// Mitsubishi GX Works2 project: Final Project   PLC: Q00U

PROGRAM CLDa
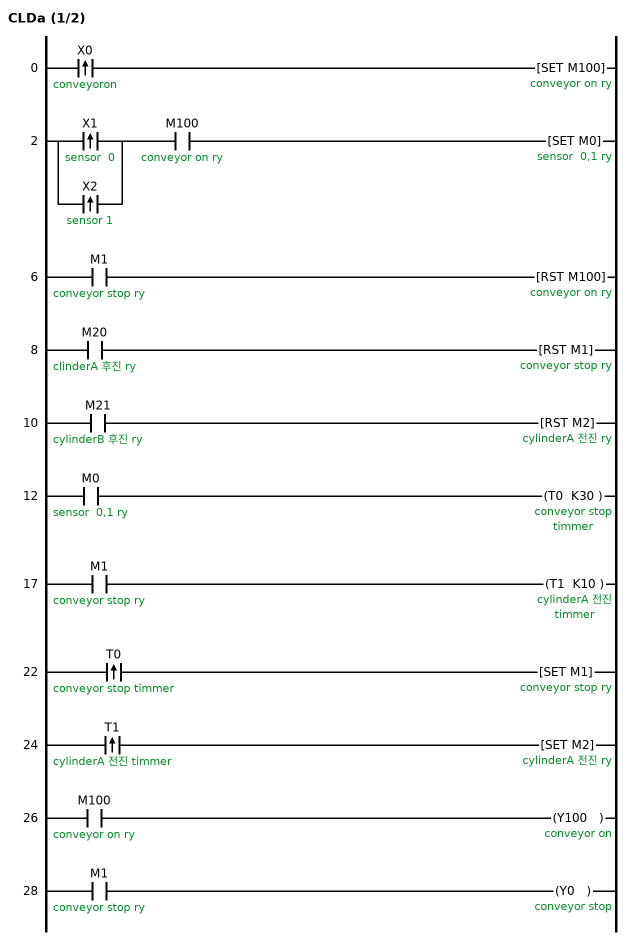
0     LDP     X0  ; conveyoron
      SET     M100  ; conveyor on ry
2     LDP     X1  ; sensor  0
      ORP     X2  ; sensor 1
      AND     M100  ; conveyor on ry
      SET     M0  ; sensor  0,1 ry
6     LD      M1  ; conveyor stop ry
      RST     M100  ; conveyor on ry
8     LD      M20  ; clinderA 후진 ry
      RST     M1  ; conveyor stop ry
10    LD      M21  ; cylinderB 후진 ry
      RST     M2  ; cylinderA 전진 ry
12    LD      M0  ; sensor  0,1 ry
      OUT     T0 K30  ; conveyor stop timmer
17    LD      M1  ; conveyor stop ry
      OUT     T1 K10  ; cylinderA 전진 timmer
22    LDP     T0  ; conveyor stop timmer
      SET     M1  ; conveyor stop ry
24    LDP     T1  ; cylinderA 전진 timmer
      SET     M2  ; cylinderA 전진 ry
26    LD      M100  ; conveyor on ry
      OUT     Y100  ; conveyor on
28    LD      M1  ; conveyor stop ry
      OUT     Y0  ; conveyor stop
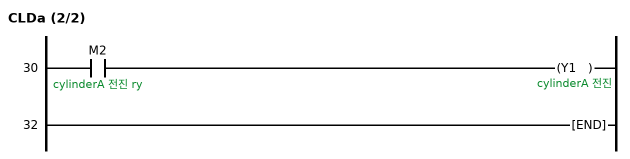
30    LD      M2  ; cylinderA 전진 ry
      OUT     Y1  ; cylinderA 전진
32    END
END_PROGRAM

PROGRAM sensor1
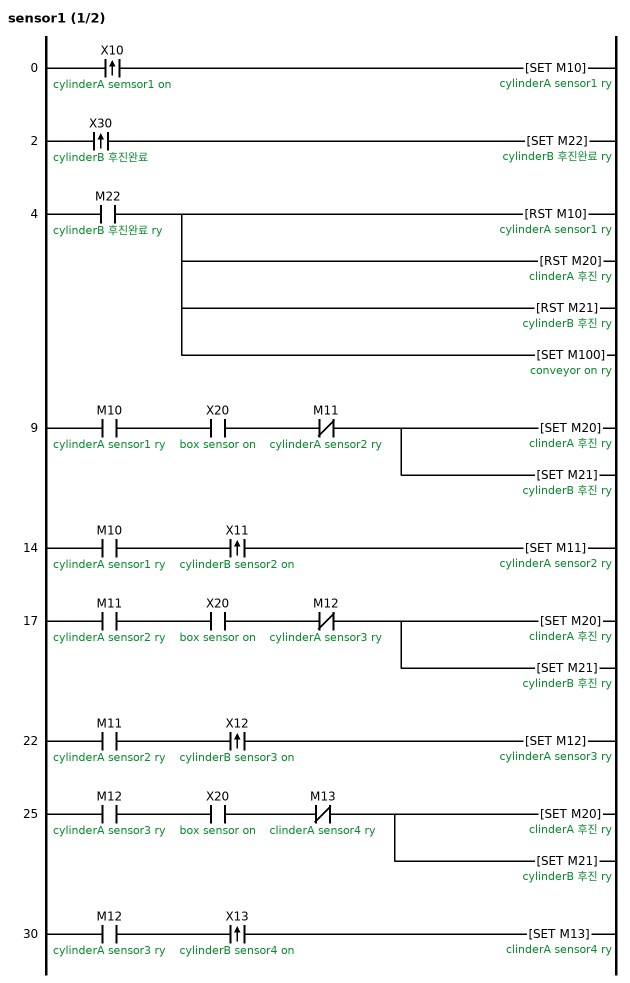
0     LDP     X10  ; cylinderA semsor1 on
      SET     M10  ; cylinderA sensor1 ry
2     LDP     X30  ; cylinderB 후진완료
      SET     M22  ; cylinderB 후진완료 ry
4     LD      M22  ; cylinderB 후진완료 ry
      RST     M10  ; cylinderA sensor1 ry
      RST     M20  ; clinderA 후진 ry
      RST     M21  ; cylinderB 후진 ry
      SET     M100  ; conveyor on ry
9     LD      M10  ; cylinderA sensor1 ry
      AND     X20  ; box sensor on
      ANI     M11  ; cylinderA sensor2 ry
      SET     M20  ; clinderA 후진 ry
      SET     M21  ; cylinderB 후진 ry
14    LD      M10  ; cylinderA sensor1 ry
      ANDP    X11  ; cylinderB sensor2 on
      SET     M11  ; cylinderA sensor2 ry
17    LD      M11  ; cylinderA sensor2 ry
      AND     X20  ; box sensor on
      ANI     M12  ; cylinderA sensor3 ry
      SET     M20  ; clinderA 후진 ry
      SET     M21  ; cylinderB 후진 ry
22    LD      M11  ; cylinderA sensor2 ry
      ANDP    X12  ; cylinderB sensor3 on
      SET     M12  ; cylinderA sensor3 ry
25    LD      M12  ; cylinderA sensor3 ry
      AND     X20  ; box sensor on
      ANI     M13  ; clinderA sensor4 ry
      SET     M20  ; clinderA 후진 ry
      SET     M21  ; cylinderB 후진 ry
30    LD      M12  ; cylinderA sensor3 ry
      ANDP    X13  ; cylinderB sensor4 on
      SET     M13  ; clinderA sensor4 ry
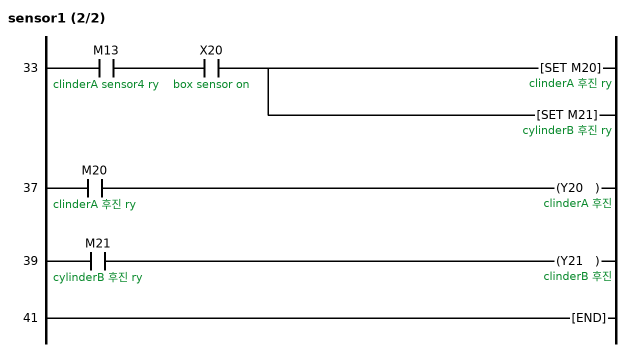
33    LD      M13  ; clinderA sensor4 ry
      AND     X20  ; box sensor on
      SET     M20  ; clinderA 후진 ry
      SET     M21  ; cylinderB 후진 ry
37    LD      M20  ; clinderA 후진 ry
      OUT     Y20  ; clinderA 후진
39    LD      M21  ; cylinderB 후진 ry
      OUT     Y21  ; clinderB 후진
41    END
END_PROGRAM

PROGRAM M10
0     END
END_PROGRAM
